// TIA Portal project "babu_PushButtonDualStateHMI" (V15)

(* hardware
DEVICE "S7-1200 station_1"  S7-1200 Station
   slot 0: "Rack_0"  S7-1200 Rack  Rack  V1.0
   slot 1: "PLC_1"  CPU 1214C DC/DC/DC  6ES7 214-1AG40-0XB0  V4.2
DEVICE "HMI_1"  KTP400 Basic PN
   slot 0: "HMI_1"  KTP400 Basic PN  6AV2 123-2DB03-0AX0  15.0.0.0
   slot 1: "HMI_RT_1"  KTP400 Basic PN  6AV2 123-2DB03-0AX0  15.0.0.0
   slot 5: "HMI_1.IE_CP_1"  PROFINET Interface  15.0.0.0
      slot 1: "PROFINET Interface_1"  PROFINET Interface
         slot 1: "Port_1"  Port
*)

// ===== PLC "PLC_1"  CPU 1214C DC/DC/DC =====

VAR_GLOBAL   // PLC tag table "Default tag table"
   "PUSH BUTTON" AT %M0.0 : Bool;
   "PUSH BUTTON MEM" AT %M0.1 : Bool;
   "PUSH BUTTON PREV STATE" AT %M0.2 : Bool;
   "PUSH BUTTON CURRENT STATE" AT %M0.3 : Bool;
   "MOTOR" AT %Q0.0 : Bool;
END_VAR

ORGANIZATION_BLOCK "Main"   // OB1, LAD, ProgramCycle
TITLE = "Main Program Sweep (Cycle)"
{ S7_Optimized_Access := 'TRUE' }
VERSION : 0.1
   VAR_INPUT
      Initial_Call : Bool;   // Initial call of this OB
      Remanence : Bool;   // =True, if remanent data are available
   END_VAR
   VAR_TEMP   // added for the SCL form of the ladder/FBD networks
      _w1 : Bool;
   END_VAR
BEGIN

REGION Network 1
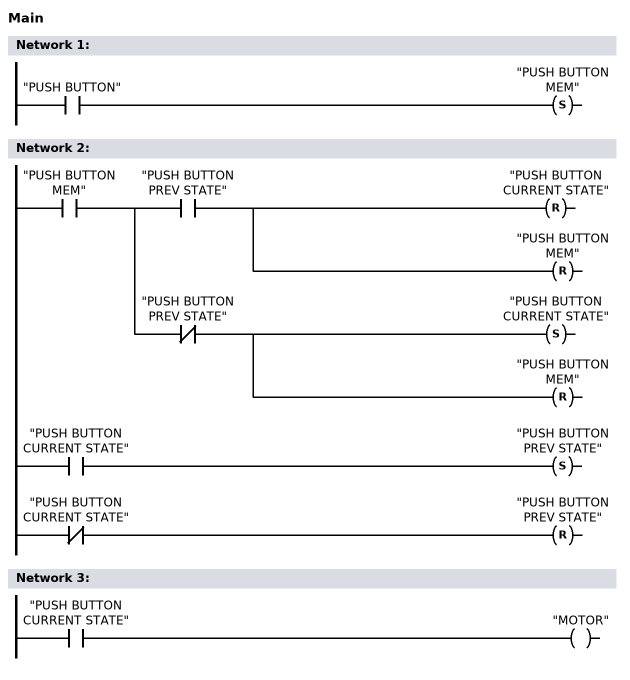
   RUNG wire#powerrail
      Contact( "PUSH BUTTON" )
      S_Coil( "PUSH BUTTON MEM" )
   END_RUNG
   // the same network as SCL:
   IF "PUSH BUTTON" THEN "PUSH BUTTON MEM" := TRUE; END_IF;
END_REGION

REGION Network 2
   RUNG wire#powerrail
      Contact( "PUSH BUTTON MEM" )
      wire#w1
      Contact( "PUSH BUTTON PREV STATE" )
      wire#w2
      R_Coil( "PUSH BUTTON CURRENT STATE" )
   END_RUNG
   RUNG wire#w2
      R_Coil( "PUSH BUTTON MEM" )
   END_RUNG
   RUNG wire#w1
      I_Contact( "PUSH BUTTON PREV STATE" )
      wire#w3
      S_Coil( "PUSH BUTTON CURRENT STATE" )
   END_RUNG
   RUNG wire#w3
      R_Coil( "PUSH BUTTON MEM" )
   END_RUNG
   RUNG wire#powerrail
      Contact( "PUSH BUTTON CURRENT STATE" )
      S_Coil( "PUSH BUTTON PREV STATE" )
   END_RUNG
   RUNG wire#powerrail
      I_Contact( "PUSH BUTTON CURRENT STATE" )
      R_Coil( "PUSH BUTTON PREV STATE" )
   END_RUNG
   // the same network as SCL:
   IF "PUSH BUTTON MEM" AND "PUSH BUTTON PREV STATE" THEN "PUSH BUTTON CURRENT STATE" := FALSE; END_IF;
   #_w1 := "PUSH BUTTON MEM";
   IF "PUSH BUTTON MEM" AND "PUSH BUTTON PREV STATE" THEN "PUSH BUTTON MEM" := FALSE; END_IF;
   IF #_w1 AND NOT "PUSH BUTTON PREV STATE" THEN
       "PUSH BUTTON CURRENT STATE" := TRUE;
       "PUSH BUTTON MEM" := FALSE;
   END_IF;
   IF "PUSH BUTTON CURRENT STATE" THEN "PUSH BUTTON PREV STATE" := TRUE; END_IF;
   IF NOT "PUSH BUTTON CURRENT STATE" THEN "PUSH BUTTON PREV STATE" := FALSE; END_IF;
END_REGION

REGION Network 3
   RUNG wire#powerrail
      Contact( "PUSH BUTTON CURRENT STATE" )
      Coil( "MOTOR" )
   END_RUNG
   // the same network as SCL:
   "MOTOR" := "PUSH BUTTON CURRENT STATE";
END_REGION
END_ORGANIZATION_BLOCK

(* ===== HMI "HMI_RT_1" =====
connection "HMI_Connection_1": ETHERNET, SMART_S7_1200_OMS

HMI tags "Default tag table"
   "PUSH BUTTON CURRENT STATE" : Bool = PLC "PUSH BUTTON CURRENT STATE" AT %M0.3, 1 s
   "PUSH BUTTON" : Bool = PLC "PUSH BUTTON" AT %M0.0, 1 s
   "PUSH BUTTON MEM" : Bool = PLC "PUSH BUTTON MEM" AT %M0.1, 1 s

screen "Root screen" 480x272, template "Template_1"
   Switch "Pushbutton_Round_G" at 1,2 size 68x62; CaptionText 'Switch'; TextOff '0'; TextOn '1'; PictureOff "Pushbutton_Round_G_Off_256c"; PictureOn "Pushbutton_Round_G_On_256c"
      ProcessValue <- "PUSH BUTTON"
   GraphicView "Graphic view_3" at 319,18 size 89x79; Picture "Graphic_3"
      Appearance <- "PUSH BUTTON CURRENT STATE"
   GraphicIOField "PlotLight_Round_R" at 1,64 size 68x62; PictureOn "PilotLight_Round_R_On_256c"; PictureOff "PilotLight_Round_R_Off_256c"
*)